FUNCTION_BLOCK DateAndTimePointerComparer EXTENDS Object IMPLEMENTS IPointerComparer
VAR
	_ClassName : STRING := __POUNAME();
END_VAR

{attribute 'monitoring' := 'call'}
PROPERTY ClassName : STRING
GET
ClassName := _ClassName;
END_GET
END_PROPERTY

{attribute "object_name" := "Compare"}
METHOD Compare : COMPARISION_RESULT
VAR_INPUT
	left : PVOID;
	right : PVOID;
END_VAR
VAR
	leftPointer : POINTER TO DATE_AND_TIME; 
	rightPointer : POINTER TO DATE_AND_TIME; 
END_VAR
IF left = 0 AND right = 0 THEN
	Compare := COMPARISION_RESULT.EQUALS;
	RETURN;
END_IF

IF left = 0 THEN
	Compare := COMPARISION_RESULT.LEFT_LESS_RIGHT;
	RETURN;	
END_IF

IF right = 0 THEN
	Compare := COMPARISION_RESULT.LEFT_GREATER_RIGHT;
	RETURN;	
END_IF

leftPointer := left;
rightPointer := right;

IF leftPointer^ < rightPointer^ THEN
	Compare := COMPARISION_RESULT.LEFT_LESS_RIGHT;
ELSIF leftPointer^ > rightPointer^ THEN
	Compare := COMPARISION_RESULT.LEFT_GREATER_RIGHT;
ELSE
	Compare := COMPARISION_RESULT.EQUALS;	
END_IF
END_METHOD

{attribute 'monitoring' := 'call'}
PROPERTY Size : ULINT
GET
Size := XSIZEOF(THIS^);
END_GET
END_PROPERTY

END_FUNCTION_BLOCK

(* stored: Version 1.1.0.1
   POU DateAndTimePointerComparer: Id {32cc5146-52ad-4380-a621-cba410028ddf}, SpecialFunc None
   Property ClassName: Id {3f714cb9-a97c-48c0-9482-2bfd7260a4d1}
   Get Get: Id {d84295e8-1019-4e08-a08a-7b7ef668d8b9}
   Method Compare: Id {7ffc095d-817e-4531-88c5-5ca45ce1fb0d}
   Property Size: Id {360da165-16ec-49a8-8e04-585859b1409c}
   Get Get: Id {95080178-4590-4b1b-aaa5-415609c7b2eb} *)
